//{attribute 'qualified_only'}
VAR_GLOBAL
	gWebAxes:		WebAxes_typ;	
END_VAR

(* stored: Version 1.1.0.1, ProductVersion 3.1.4024.3
   GVL AxesList: Id {a1d1e217-019b-0169-2c97-d10adf46ef42} *)
